PROGRAM HMI
VAR
	Loader_Name				: ARRAY [1..100] OF STRING;
	Loader_Number			: ARRAY [1..100] OF WORD;
	Loader_Status			: ARRAY [1..100] OF WORD;
	Loader_HMI_Status		: ARRAY [1..100] OF WORD;
	Loader_Last_Time		: ARRAY [1..100] OF WORD;
	Loader_Prop				: ARRAY [1..100] OF WORD;
	Loader_Exist			: ARRAY [1..100] OF BOOL;
END_VAR

// NETWORK 1

END_PROGRAM

(* stored: Version 1.1.0.1, ProductVersion 3.1.4024.13
   POU HMI: Id {c1fd9fc7-cb04-4da5-97b1-8a0fd04c1bc5}, SpecialFunc None *)
